INTERFACE IRecordDataQueue

PROPERTY PUBLIC data_def_structure_name : Tc2_System.T_MaxString
GET
END_GET
SET
END_SET
END_PROPERTY

// Record data body that is converted to T_Arg type. 
PROPERTY PUBLIC data_pointer : T_Arg
GET
END_GET
SET
END_SET
END_PROPERTY

// Measurement name of influxDB.
PROPERTY PUBLIC db_table_name : Tc2_System.T_MaxString
GET
END_GET
SET
END_SET
END_PROPERTY

// current index of data buffer.
PROPERTY PUBLIC index : UDINT
GET
END_GET
SET
END_SET
END_PROPERTY

(*
Mininum chunk record count for dynamic insert.

The cyclic data are accumulated to data buffe. When num of data in this buffer reached this specified size, these accumulated data is queued in command buffer for insert to InfluxDB.  

The chunk size will be dynamically expanded when the throughput of command queue is slowed down.
*)

PROPERTY PUBLIC minimum_chunk_size : UDINT
GET
END_GET
SET
END_SET
END_PROPERTY

// 
PROPERTY PUBLIC upper_bound_of_data_buffer : UDINT
GET
END_GET
SET
END_SET
END_PROPERTY

END_INTERFACE

(* stored: Version 1.1.0.1, ProductVersion 3.1.4024.12
   Itf IRecordDataQueue: Id {31172c77-633a-46d5-b927-3b44dc9446a9}
   Property data_def_structure_name: Id {272557a6-6b2c-4c63-901b-84e0e6d9e8fe}
   Get Get: Id {5ce1eade-bf64-47ea-91d7-941e55f3dbe8}
   Set Set: Id {44dc5f52-8a64-451c-9a47-a26c1e50a769}
   Property data_pointer: Id {77a45e8f-03a6-4d52-b9fe-4d82ddf16572}
   Get Get: Id {b5b5edb7-cfc2-4776-9736-ef572981e8c6}
   Set Set: Id {6c42489c-6a20-4320-8860-46c5c2ba4037}
   Property db_table_name: Id {afbea261-1eab-4676-8eeb-028a28145ab2}
   Get Get: Id {f9d8cd56-ed8f-49e2-ade0-5487d7710609}
   Set Set: Id {670228aa-03dc-40cc-848b-d2232a202fc7}
   Property index: Id {0ee0c4ae-9c70-4169-961c-a0161b321b3a}
   Get Get: Id {ac706858-0c73-4513-96a2-c46f956b5591}
   Set Set: Id {3544b6c6-76b1-4bf0-8e21-1e23c1255461}
   Property minimum_chunk_size: Id {42e269e0-c904-48ea-a9c1-9c6264540f8d}
   Get Get: Id {8f120c89-228e-4a85-b036-9e808e093df5}
   Set Set: Id {f594dc65-1837-4093-beba-672bbcbcc1c7}
   Property upper_bound_of_data_buffer: Id {561f1f89-809b-4fcc-ae97-102637f1dae1}
   Get Get: Id {0972a6d0-c774-4c4e-84b1-a73b0cd738b4}
   Set Set: Id {738dbc58-d380-444d-8c86-8ac2b3ed6832} *)
